# EPICS substitutions: BLDApp/Db/IOC-SYS0-BD01bsa.substitutions
#==============================================================================
#
# Abs:  LCLS Beam Synchronous Acquisition records for SYS0 BD01
#
# Name: IOC-SYS0-BD01bsa.substitutions
#
# Associated Displays: bsa_sys0_maint.edl
#
# Rem:  Instantiate one line for every beam synchronous item.
#
# Macros:
#	DEVICE	Name of the beam synchronous triggered device.  Must match the
#		name in <ioc>trig.substitutions without the 3rd colon and beyond.
#	LOC	IOC location.
#	UN	IOC unit number.
#	IOC	Name of IOC that contains the EVR, not including the 3rd colon.
#	ATRB    BSA attribute name
#	IN	Input to BSA record
#	SLCLNK	Set to "" if the IOC is not slc-aware.
#		Otherwise, set to "<device>:FANOUTSLC".
#==============================================================================
#
file bsaBLDEdef.db {
    pattern
    { DEVICE, LOC, UN, SLCLNK }
    { BLD:SYS0:500, SYS0, 500, "" }
}

file bsaBLDReceiverPhaseCavityEdef.db {
    pattern
    { DEVICE, LOC, UN, SLCLNK }
    { BLD:SYS0:500, SYS0, 500, "" }
}
